INTERFACE I_Device

METHOD turnOff
VAR_INPUT
END_VAR
END_METHOD

METHOD turnOn
VAR_INPUT
END_VAR
END_METHOD

END_INTERFACE

(* stored: Version 1.1.0.1
   Itf I_Device: Id {d265e15a-2850-4254-a94a-1abeae43410c}
   Method turnOff: Id {f1a75f6c-4a4f-4aa4-b3a0-6d4395d6e808}
   Method turnOn: Id {48516bab-8eef-4821-aa55-b9c684cdb512} *)
